TYPE ST_RingBuffer :
STRUCT
	Table		: ARRAY [0..3599] OF LREAL;
END_STRUCT
END_TYPE

(* stored: Version 1.1.0.1, ProductVersion 3.1.4024.9
   DUT ST_RingBuffer: Id {9e8929aa-43a5-4b53-9519-1ff5e7b96212} *)
